// SIMATIC S7-200 project (STEP 7-Micro/WIN), CPU 226 REL 01.23

ORGANIZATION_BLOCK MAIN:OB1
TITLE=程序注释
BEGIN
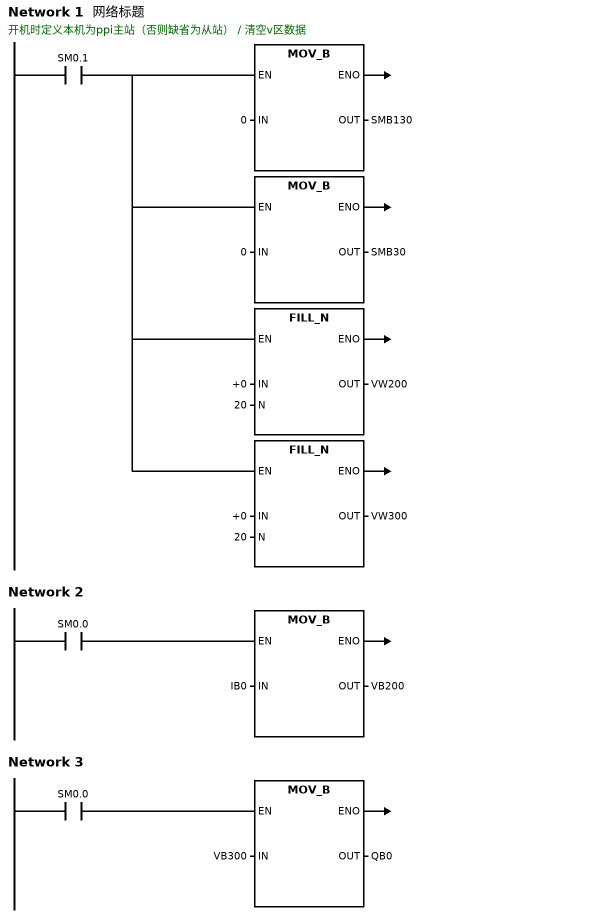
Network 1 // 网络标题
// 开机时定义本机为ppi主站（否则缺省为从站）
// 清空v区数据
LD     SM0.1
MOVB   0, SMB130
MOVB   0, SMB30
FILL   +0, VW200, 20
FILL   +0, VW300, 20
Network 2
LD     SM0.0
MOVB   IB0, VB200
Network 3
LD     SM0.0
MOVB   VB300, QB0
END_ORGANIZATION_BLOCK
